TYPE E_ValueType :
(
	TYPE_NOT_SPECIFIED := 0,
	TYPE_SINT := 1,
	TYPE_INT := 2,
	TYPE_DINT := 3,
	TYPE_USINT := 4,
	TYPE_UINT := 5,
	TYPE_UDINT := 6,
	TYPE_STRING := 7
) USINT;
END_TYPE

(* stored: Version 1.1.0.1, ProductVersion 3.1.0.36
   DUT E_ValueType: Id {6f842dbb-3775-4e86-b994-8b7685675dab} *)
